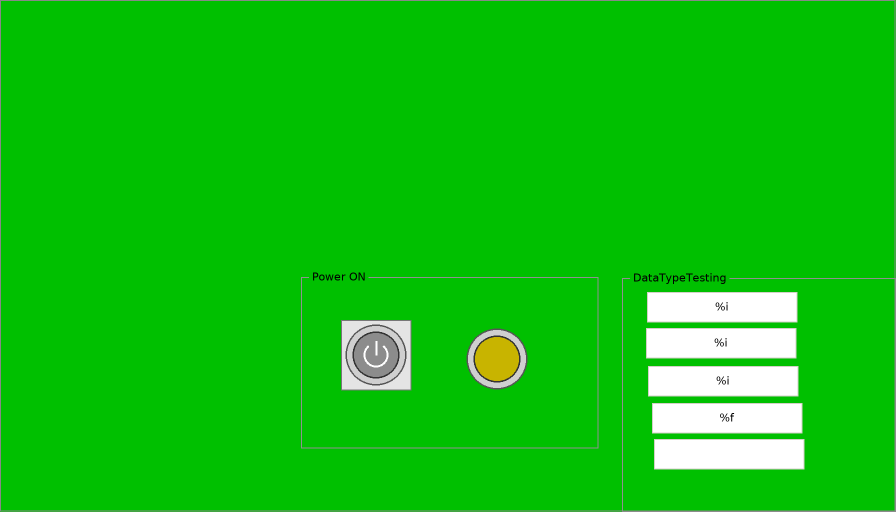
VISUALIZATION HMI  // 896x512
    GroupBox (301,269 297x179), "Power ON"
        PowerSwitch (40,51 70x70), variable: MAIN.bStart, behaviour: TOGGLE, style: Switch-PowerSwitch-Gray
        Lamp1 (161,55 70x70), variable: MAIN.bEnable, style: Lamp-Lamp1-Yellow
    GroupBox (622,270 274x242), "DataTypeTesting"
        Textfield (24,58 150x30), "%i", text variable: MAIN.nINT
        Textfield (26,96 150x30), "%i", text variable: MAIN.nUNIT
        Textfield (25,22 150x30), "%i", text variable: MAIN.bEnable
        Textfield (30,133 150x30), "%f", text variable: MAIN.fREAL
            OnMouseDown: write the text variable via Default
    Textfield (654,439 150x30)
END_VISUALIZATION

(* stored: Version 1.1.0.1, ProductVersion 3.1.4024.12
   Visu HMI: Id {d343a843-436a-4d2c-b474-0d7705f518b7} *)
